(* Logix 5000 project; controller PLC2_Project_3 Emulate 5570 rev 20.11; software revision 20.00 *)

TASK MainTask (continuous, watchdog 500 ms) : MainProgram

MODULES
   Local : Emulate 5570 (ICP 1, rev 20.11)
END_MODULES

PROGRAM MainProgram   (* main routine MainRoutine *)
VAR
   CleanTempData : BOOL;
   Item_123_Qty : DINT;
   Item_456_Qty : DINT;
   Item_789_Qty : DINT;
   Material_AddSubtract : DINT;
   Material_ID : DINT;
   Material_Qty : DINT;
   String_BarcodeInput : STRING;
   String_Null : STRING;
   String_Sort_Bit : BOOL;
   Temo_Qty : STRING;
   Temp_Direction : STRING;   // 0 = Subtraction 1 = Addition
   Temp_ID : STRING;
END_VAR

ROUTINE MainRoutine   (* ladder *)
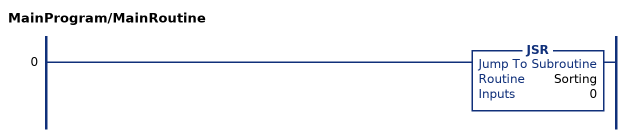
   0: JSR(Sorting,0);
END_ROUTINE

ROUTINE Sorting   (* ladder *)
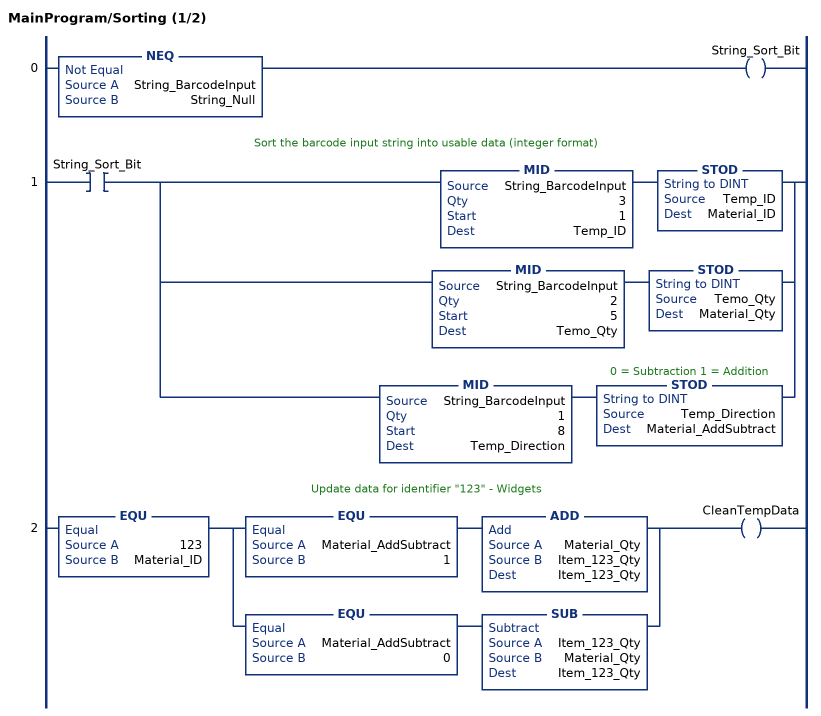
   0: NEQ(String_BarcodeInput,String_Null)OTE(String_Sort_Bit);
   // Sort the barcode input string into usable data (integer format)
   1: XIC(String_Sort_Bit)[MID(String_BarcodeInput,3,1,Temp_ID) STOD(Temp_ID,Material_ID) ,MID(String_BarcodeInput,2,5,Temo_Qty) STOD(Temo_Qty,Material_Qty) ,MID(String_BarcodeInput,1,8,Temp_Direction) STOD(Temp_Direction,Material_AddSubtract) ];
   // Update data for identifier "123" - Widgets
   2: EQU(123,Material_ID)[EQU(Material_AddSubtract,1) ADD(Material_Qty,Item_123_Qty,Item_123_Qty) ,EQU(Material_AddSubtract,0) SUB(Item_123_Qty,Material_Qty,Item_123_Qty) ]OTE(CleanTempData);
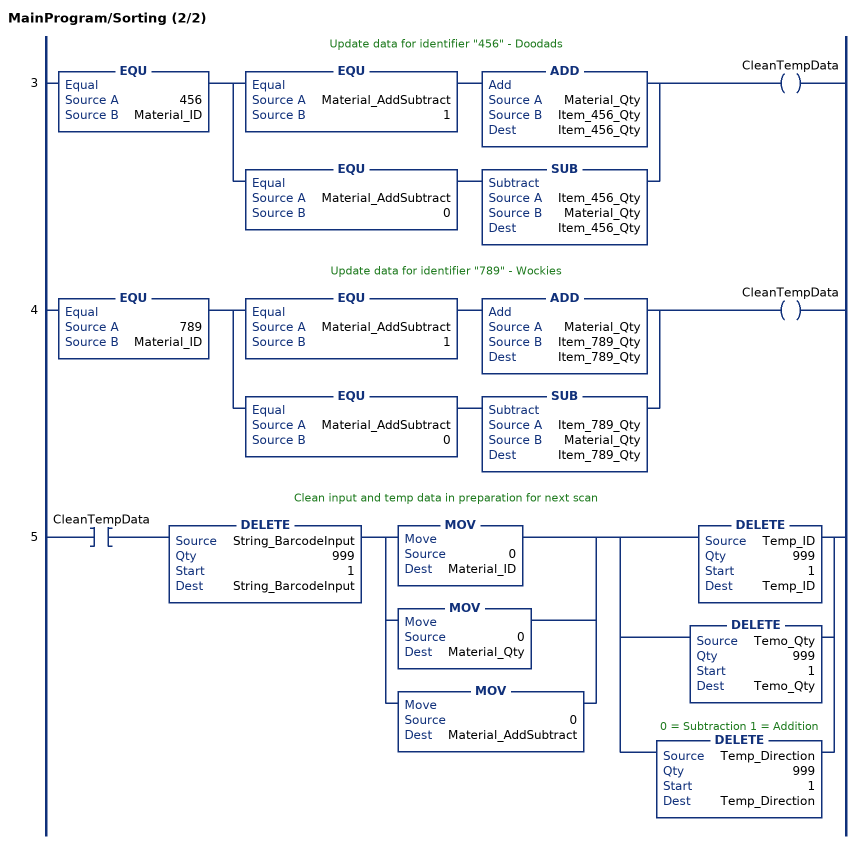
   // Update data for identifier "456" - Doodads
   3: EQU(456,Material_ID)[EQU(Material_AddSubtract,1) ADD(Material_Qty,Item_456_Qty,Item_456_Qty) ,EQU(Material_AddSubtract,0) SUB(Item_456_Qty,Material_Qty,Item_456_Qty) ]OTE(CleanTempData);
   // Update data for identifier "789" - Wockies
   4: EQU(789,Material_ID)[EQU(Material_AddSubtract,1) ADD(Material_Qty,Item_789_Qty,Item_789_Qty) ,EQU(Material_AddSubtract,0) SUB(Item_789_Qty,Material_Qty,Item_789_Qty) ]OTE(CleanTempData);
   // Clean input and temp data in preparation for next scan
   5: XIC(CleanTempData)DELETE(String_BarcodeInput,999,1,String_BarcodeInput)[MOV(0,Material_ID) ,MOV(0,Material_Qty) ,MOV(0,Material_AddSubtract) ][DELETE(Temp_ID,999,1,Temp_ID) ,DELETE(Temo_Qty,999,1,Temo_Qty) ,DELETE(Temp_Direction,999,1,Temp_Direction) ];
END_ROUTINE
END_PROGRAM
